// TIA Portal V17 export
// export: Created 2023-04-04T13:27:29.1774789Z, ExportSetting WithDefaults, DisplayName Totally Integrated Automation Portal, DisplayVersion V17, DisplayName TIA Portal Openness, DisplayVersion V17, DisplayName TIA Portal Version Control Interface, DisplayVersion V17, DisplayName STEP 7 Professional, DisplayVersion V17, DisplayName STEP 7 Safety, DisplayVersion V17, DisplayName WinCC Advanced, DisplayVersion V17
DATA_BLOCK "Queue"   // DB46
{ S7_Optimized_Access := 'TRUE' }
VERSION : 0.1
// stored: AutoNumber true, DBAccessibleFromOPCUA true, DBAccessibleFromWebserver true, IsOnlyStoredInLoadMemory false, IsRetainMemResEnabled false, IsWriteProtectedInAS false, MemoryReserve 100
   VAR RETAIN
      Queue : Array[0.."Ci_Queue_Length"] of "typ_Order_Workpiece_Buttons";
      i_Queue_Index { S7_SetPoint := 'True'} : Int;   // Index where next element will be written
      x_Queue_Full : Bool;
   END_VAR
BEGIN
END_DATA_BLOCK
